Staubli VAL3: insertItem.pgx

public program insertItem(InstrItem& x_sItem[], num x_nIndex)
  local num l_sItem
begin
  if x_nIndex<=0
    x_nIndex=0
  else
    insert(pEdit.iEvent[x_nIndex])
  endIf
  call setItem(x_sItem,x_nIndex)
end
